PROGRAM MAIN_Events
VAR
END_VAR

END_PROGRAM

(* stored: Version 1.1.0.1, ProductVersion 3.1.4024.15
   POU MAIN_Events: Id {7a39f841-be4d-45aa-93ed-4769dfe66808}, SpecialFunc None *)
